FUNCTION TFPalletizerIsCodeAssigned : BOOL
VAR_INPUT
	WorkArea : POINTER TO ARRAY [1..MAXAREA] OF TFMachinePalletizer_WorkArea;
	WorkAreaState : POINTER TO ARRAY [1..MAXAREA] OF TFMachinePalletizer_WorkAreaState;
	Code : INT;
END_VAR
VAR
	wa : INT;
	n : INT;
END_VAR

TFPalletizerIsCodeAssigned := FALSE; 

FOR wa:=1 TO MAXAREA DO
	IF WorkArea^[wa].Enable = 1 THEN
		(* Verifico se il codice è già stato assegnato *)
		IF WorkArea^[wa].Code = Code AND Code <> 0 THEN
			(* Verifico se la piazzola è in lavorazione *)
			(* Se è in lavorazione allora è inutile assegnarne un'altra con lo stesso codice *)
			IF WorkAreaState^[wa].State < WORKAREA_STATE_OCCUPIED_WORKED AND 
				WorkAreaState^[wa].State > WORKAREA_STATE_FREE_DISABLED THEN
				TFPalletizerIsCodeAssigned := TRUE;
				RETURN;
			END_IF
		END_IF
	END_IF
END_FOR

END_FUNCTION

(* stored: Version 1.1.0.1, ProductVersion 3.1.4024.11
   POU TFPalletizerIsCodeAssigned: Id {40bfd9b8-6eaa-44ce-8c1c-73f0aaa2686e}, SpecialFunc None *)
